{attribute 'linkalways'} 
{attribute 'no_explicit_call' := 'This FB is a CLASS and must be accessed using methods or properties'}
{attribute 'enable_dynamic_creation'}
FUNCTION_BLOCK AsyncResponseSessionDataProxy EXTENDS Disposable IMPLEMENTS I_AsyncResponseSessionData
VAR
	sessionStorage : I_SessionStorage;
	sessionId : T_MAXSTRING;
	responseId : T_MAXSTRING;
END_VAR

METHOD PUBLIC Error
VAR_INPUT
	Message : T_MAXSTRING;
END_VAR
VAR
	asyncReponseSessionData : I_AsyncResponseSessionData;
END_VAR
IF NOT TryGetAsyncResponseSessionData(asyncReponseSessionData) THEN
	RETURN;
END_IF

asyncReponseSessionData.Error(Message);
END_METHOD

METHOD FB_init : BOOL
VAR_INPUT
	bInitRetains : BOOL; // if TRUE, the retain variables are initialized (warm start / cold start)
	bInCopyCode : BOOL;  // if TRUE, the instance afterwards gets moved into the copy code (online change)
	SessionStorage : I_SessionStorage;
	SessionId : T_MAXSTRING;
	ResponseId : T_MAXSTRING;
END_VAR
THIS^.sessionStorage := SessionStorage;
THIS^.sessionId := SessionId;
THIS^.responseId := ResponseId;
END_METHOD

PROPERTY PUBLIC IsPending : BOOL
GET
VAR
	asyncReponseSessionData : I_AsyncResponseSessionData;
END_VAR
IF NOT TryGetAsyncResponseSessionData(asyncReponseSessionData) THEN
	RETURN;
END_IF

IsPending := asyncReponseSessionData.IsPending;
END_GET
END_PROPERTY

METHOD PUBLIC Success
VAR_INPUT
END_VAR
VAR
	asyncReponseSessionData : I_AsyncResponseSessionData;
END_VAR
IF NOT TryGetAsyncResponseSessionData(asyncReponseSessionData) THEN
	RETURN;
END_IF

asyncReponseSessionData.Success();
END_METHOD

METHOD PUBLIC SuccessWithPayload
VAR_INPUT
	PayloadDataAddress : PVOID;
	PayloadDataSize : UDINT;
END_VAR
VAR
	asyncReponseSessionData : I_AsyncResponseSessionData;
END_VAR
IF NOT TryGetAsyncResponseSessionData(asyncReponseSessionData) THEN
	RETURN;
END_IF

asyncReponseSessionData.SuccessWithPayload(PayloadDataAddress, PayloadDataSize);
END_METHOD

PROPERTY PUBLIC SuggestedRetryDelayInMs : UDINT
GET
VAR
	asyncReponseSessionData : I_AsyncResponseSessionData;
END_VAR
IF NOT TryGetAsyncResponseSessionData(asyncReponseSessionData) THEN
	RETURN;
END_IF

SuggestedRetryDelayInMs := asyncReponseSessionData.SuggestedRetryDelayInMs;
END_GET
SET // PUBLIC
VAR
	asyncReponseSessionData : I_AsyncResponseSessionData;
END_VAR
IF NOT TryGetAsyncResponseSessionData(asyncReponseSessionData) THEN
	RETURN;
END_IF

asyncReponseSessionData.SuggestedRetryDelayInMs := SuggestedRetryDelayInMs;
END_SET
END_PROPERTY

METHOD PROTECTED TryGetAsyncResponseSessionData : BOOL;
VAR_INPUT
	Destination : REFERENCE TO I_AsyncResponseSessionData;
END_VAR
VAR
	sessionData : I_SessionData;
	asyncSessionData : I_AsyncResponseSessionData;
END_VAR
IF NOT sessionStorage.TryRetreiveSessionDataById(sessionId, responseId, sessionData) THEN
	RETURN;
END_IF

IF NOT __QUERYINTERFACE(sessionData, asyncSessionData) THEN
	RETURN;
END_IF

Destination := asyncSessionData;
TryGetAsyncResponseSessionData := TRUE;
END_METHOD

METHOD PUBLIC TryUpdateServerResponse : BOOL
VAR_INPUT
	Response : I_ServerResponse;
END_VAR
VAR
	asyncReponseSessionData : I_AsyncResponseSessionData;
END_VAR
IF NOT TryGetAsyncResponseSessionData(asyncReponseSessionData) THEN
	RETURN;
END_IF

TryUpdateServerResponse := asyncReponseSessionData.TryUpdateServerResponse(Response);
END_METHOD

END_FUNCTION_BLOCK

(* stored: Version 1.1.0.1, ProductVersion 3.1.4024.12
   POU AsyncResponseSessionDataProxy: Id {bcb02eb0-e014-04b5-02eb-09be8f08cf5b}, SpecialFunc None
   Folder Constructor: Id {b5d74c72-0e88-01d6-37c0-27d10659248f}
   Folder Protected: Id {b38f42b2-9624-05db-355c-ea3eaf9212c6}
   Method Error: Id {fcc6a772-3725-0f26-318c-a24a3405422e}
   Method FB_init: Id {211ec0f6-35b8-0342-27a3-6a265a16fe1f}
   Property IsPending: Id {6cf1f764-c7d3-0720-0365-c0c3f2cb9025}
   Get Get: Id {fb2892d3-d077-0a73-1a45-a33f2d011f9a}
   Method Success: Id {2e3c2832-2fa2-0d30-084d-bcf44ae0a1e5}
   Method SuccessWithPayload: Id {63f145b2-03c4-0151-1d0f-135bd8f0f833}
   Property SuggestedRetryDelayInMs: Id {a5c0c372-b7bc-007b-11cf-8c5d9698d5fb}
   Get Get: Id {471a2864-443e-0278-1822-e2d0943e3c01}
   Set Set: Id {dcbc7674-a243-0716-0e8c-0eba6807595a}
   Method TryGetAsyncResponseSessionData: Id {43ec3982-729f-0294-2d5c-a288a75095f3}
   Method TryUpdateServerResponse: Id {439ceb7d-1235-0621-39a4-131e3cc2448f} *)
